Fanuc KAREL source: kb00176.KL

-- PROVISIONAL review KL for V940-1; original PC SHA256 038b1df6ecfa2b0f046625b1a8de315f9255eb0aff05e9aec2de7f76913311f7
-- Incomplete behavior may be omitted. Consult companion uncertainty JSON. Do not deploy.
PROGRAM KB00176
%NOLOCKGROUP
BEGIN
  -- V9_ZERO_TABLE_METADATA_HINT layout=0002_ascii; no indexed target words; source/name/runtime held
  -- UNRESOLVED_PC offsets 5-12; opcodes 9D,23
  -- UNRESOLVED_PC offsets 17-32; opcodes 2E,22,32,35
  -- UNRESOLVED_PC offsets 37-44; opcodes 9D,23
  -- UNRESOLVED_PC offsets 49-79; opcodes 27,22,22,1C,22,27,9D,31
  -- UNRESOLVED_PC offsets 84-88; opcodes 7F
END KB00176
